Staubli VAL3: arrayToJoint.pgx

public program arrayToJoint(num& x_nNumInput[], jointRx& x_jJointOutput[])
  local num l_nNumOutput[6]
begin

  //==========解析两个机器人之间通讯收发的数据和指令==========

  //将数组数据解析成机器人的关节位置
  l_nNumOutput=x_nNumInput

  x_jJointOutput.j1=l_nNumOutput[0]
  x_jJointOutput.j2=l_nNumOutput[1]
  x_jJointOutput.j3=l_nNumOutput[2]
  x_jJointOutput.j4=l_nNumOutput[3]
  x_jJointOutput.j5=l_nNumOutput[4]
  x_jJointOutput.j6=l_nNumOutput[5]

end
